RoboDK station: UR3_Pick_Place.rdk

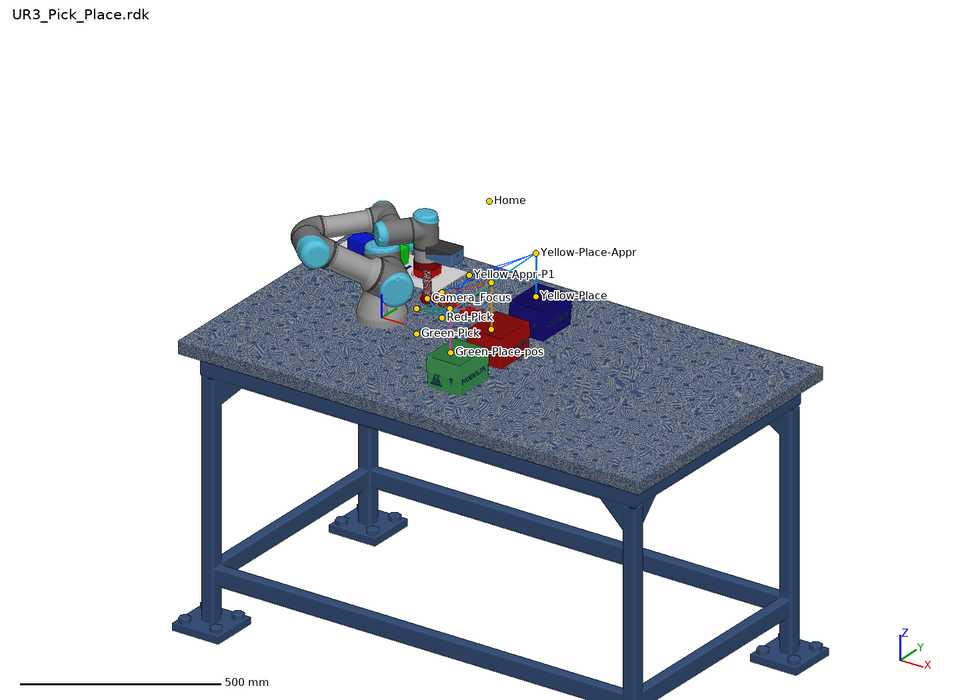
[picture v0: the station drawn from its stored meshes, robots at their saved joint values, targets as dots, program paths as lines]
Station UR3_Pick_Place (saved by RoboDK 5.4.1). Poses are relative to the parent item; angles as X-Y-Z fixed-axis rotations.
Station parameters (name, value as stored): IO_5, 1
  - frame UR3 Base at (0, 0, 0) mm
    - robot UR3: 6 axes, payload 3 kg, reach 500 mm, repeatability 0.1 mm, weight 11 kg
        modified DH rows (alpha deg, a mm, theta deg, d mm): 0, 0, 0, 151.9; 90, 0, 180, 0; 0, 243.65, 0, 0; 0, 213, 0, 110.4; -90, 0, 0, 83.4; 90, 0, 180, 82.4
        joint limits [-360, -360, -360, -360, -360, -360] to [360, 360, 360, 360, 360, 360]; home [0, -90, -90, 0, 90, 0]; saved at [48.153, -30.635, -146.156, -92.197, 88.87, 48.143]
      - tool Suction_Gripper, TCP at (0, 0, 110) mm, size 63.3 x 62.3 x 118 mm, geometry from Suction_Gripper.STEP
      - tool Camera, TCP at (0.03, -70.24, -12.53) mm, size 53 x 116 x 38 mm, geometry from Cam2D_SICK_VSPP_5F2113.sld
    - target Home (Cartesian target) at (403.4, -110.4, 478.95) mm, rotated rx -90 ry 0 rz -90 deg; joints [0, -90, -90, 0, 90, 0] of UR3
    - target Camera_Focus (Cartesian target) at (144.98, -9.29, 97.12) mm, rotated rx -178.48 ry 0 rz -90 deg; joints [48.127, -30.627, -146.695, -91.665, 88.87, 48.117] of UR3
    - target Yellow-Pick (Cartesian target) at (193.61, 104.25, 59.99) mm, rotated rx -179.29 ry 0 rz -90 deg; joints [59.044, -76.454, -144.258, -48.925, 89.395, 59.042] of UR3
    - target Yellow-Appr-P1 (Cartesian target) at (193.61, 104.25, 129.98) mm, rotated rx -179.29 ry 0 rz -90 deg; joints [59.044, -65.301, -129.223, -75.113, 89.395, 59.042] of UR3
    - target Yellow-Place (Cartesian target) at (346.96, 173.82, 85.56) mm, rotated rx -179.29 ry 0 rz -90 deg; joints [43.387, -113.771, -94.131, -61.585, 89.515, 43.384] of UR3
    - target Yellow-Place-Appr (Cartesian target) at (346.96, 173.82, 205.56) mm, rotated rx -179.29 ry 0 rz -90 deg; joints [43.389, -107.639, -68.833, -93.015, 89.515, 43.387] of UR3
    - target Red-Pick (Cartesian target) at (194.79, -15.82, 59.73) mm, rotated rx -179.29 ry 0 rz -90 deg; joints [30.172, -66.701, -149.718, -52.971, 89.645, 30.171] of UR3
    - target Red-Appr (Cartesian target) at (194.8, -15.82, 129.73) mm, rotated rx -179.29 ry 0 rz -90 deg; joints [30.173, -56.356, -133.241, -79.793, 89.645, 30.171] of UR3
    - target Red-Place-Appr (Cartesian target) at (344.8, -15.82, 199.73) mm, rotated rx -179.29 ry 0 rz -90 deg; joints [16.143, -96.634, -84.116, -88.571, 89.804, 16.142] of UR3
    - target Red-Place (Cartesian target) at (344.8, -15.82, 69.73) mm, rotated rx -179.29 ry 0 rz -90 deg; joints [16.142, -106.602, -109.753, -52.967, 89.804, 16.141] of UR3
    - target Green-Pick (Cartesian target) at (194.8, -125.82, 59.73) mm, rotated rx -179.29 ry 0 rz -90 deg; joints [-4.48, -80.711, -141.556, -47.028, 90.055, -4.48] of UR3
    - target Green-pick-aapr (Cartesian target) at (194.8, -125.82, 129.73) mm, rotated rx -179.29 ry 0 rz -90 deg; joints [-4.48, -69.374, -127.223, -72.7, 90.055, -4.48] of UR3
    - target Green-Place-pos (Cartesian target) at (348.16, -199.1, 80.31) mm, rotated rx -179.29 ry 0 rz -90 deg; joints [-13.869, -117.211, -90.452, -61.652, 90.169, -13.868] of UR3
    - target Green-place-appr (Cartesian target) at (344.79, -195.82, 199.73) mm, rotated rx -179.29 ry 0 rz -90 deg; joints [-13.51, -109.8, -67.516, -91.997, 90.165, -13.509] of UR3
    - object RoboDK Nametag Plate 500x200mm at (30, 330, 0) mm, rotated rx 0 ry 0 rz 90 deg, size 140 x 350 x 3.5 mm, geometry from RoboDK-Nametag-Plate-500x200mm.sld
  - object Table 1400x800x800 at (0, 0, 0) mm, size 1420 x 820 x 800 mm, geometry from Table-1400mmx800mmx800mm.sld
  - program Prog_Place_Blue (11 instructions, listed below)
  - program Prog_Place_Red (9 instructions, listed below)
  - program Prog_Place_Green (10 instructions, listed below)
  - camera Camera
  - program Prog_Return_Green (9 instructions, listed below)
  - program Prog_Return_Red (10 instructions, listed below)
  - program Prog_Return_Blue (8 instructions, listed below)
  - program Program_Animation (6 instructions, listed below)
  - object Blue-Box at (307.84, 115.7, 0) mm, size 109.7 x 131.2 x 86.2 mm, geometry from Box-12inx10in-Opened.sld
  - object Red-Box at (313.37, -73.28, 0) mm, size 109.7 x 131.2 x 86.2 mm, geometry from Box-12inx10in-Opened.sld
  - object Green-Box at (316.63, -256.72, 0) mm, size 109.7 x 131.2 x 86.2 mm, geometry from Box-12inx10in-Opened.sld
  - object Red-Cube at (-70, 237, 0) mm, size 50 x 50 x 50 mm, geometry from Cube-50mm.sld
  - object Blue-Cube at (-270, 237, 0) mm, size 50 x 50 x 50 mm, geometry from Cube-50mm.sld
  - object Green-Cube at (-170, 237, 0) mm, size 50 x 50 x 50 mm, geometry from Cube-50mm.sld
  - camera Camera 2
  - program Prog_Home_Pos (3 instructions, listed below)
  - program Prog_Cam_Pos (3 instructions, listed below)
  - object IDLEArea at (-40, 380, 0) mm, rotated rx 0 ry 0 rz 180 deg, size 181.5 x 27.8 x 8.8 mm, geometry from IDLEArea.STEP
  - object WorkArea at (280, 160, 0) mm, rotated rx 0 ry 0 rz 180 deg, size 271.5 x 30 x 9 mm, geometry from WorkArea.STEP
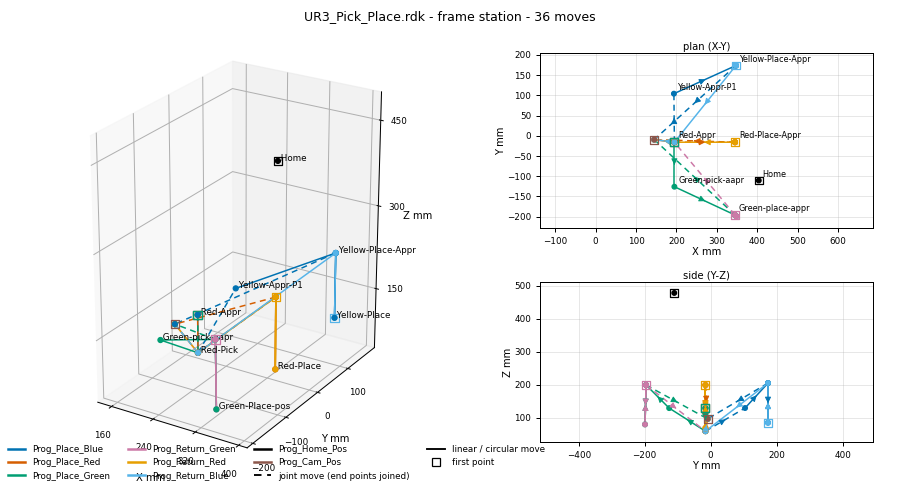
[picture p0: tool path of UR3_Pick_Place.rdk in frame station, 36 of 36 moves have a stored position in this frame; points joined in program order, loops and branches not executed]

--- program Prog_Place_Blue (robot UR3) ---
  Set Ref.: UR3 Base
  Set Tool: Gripper at (0, 0, 108) mm
  MoveJ (Red-Appr)
  MoveL (Red-Pick)
  Attach to Suction_Gripper
  MoveJ (Yellow-Appr-P1)
  MoveL (Yellow-Place-Appr)
  MoveL (Yellow-Place)
  Detach from Suction_Gripper
  MoveL (Yellow-Place-Appr)
  MoveJ (Camera_Focus)

--- program Prog_Place_Red (robot UR3) ---
  Set Ref.: UR3 Base
  MoveL (Red-Appr)
  MoveL (Red-Pick)
  Attach to Suction_Gripper
  MoveJ (Red-Place-Appr)
  MoveL (Red-Place)
  Detach from Suction_Gripper
  MoveL (Red-Place-Appr)
  MoveJ (Camera_Focus)

--- program Prog_Place_Green (robot UR3) ---
  Set Ref.: UR3 Base
  MoveL (Red-Appr)
  MoveJ (Red-Pick)
  Attach to Suction_Gripper
  MoveL (Green-pick-aapr)
  MoveL (Green-place-appr)
  MoveL (Green-Place-pos)
  Detach from Suction_Gripper
  MoveL (Green-place-appr)
  MoveJ (Camera_Focus)

--- program Prog_Return_Green (robot UR3) ---
  Set Ref.: UR3 Base
  Set Tool: Suction_Gripper
  MoveJ (Green-place-appr)
  MoveL (Green-Place-pos)
  Attach to Suction_Gripper
  MoveL (Green-place-appr)
  MoveJ (Red-Pick)
  Detach from Suction_Gripper
  MoveL (Camera_Focus)

--- program Prog_Return_Red (robot UR3) ---
  Set Ref.: UR3 Base
  Set Tool: Suction_Gripper
  MoveJ (Red-Place-Appr)
  MoveL (Red-Place)
  Attach to Suction_Gripper
  MoveL (Red-Place-Appr)
  MoveL (Red-Pick)
  Detach from Suction_Gripper
  MoveL (Camera_Focus)
  Set IO_5=1

--- program Prog_Return_Blue (robot UR3) ---
  Set Ref.: UR3 Base
  Set Tool: Suction_Gripper
  MoveJ (Yellow-Place)
  Attach to Suction_Gripper
  MoveL (Yellow-Place-Appr)
  MoveL (Red-Pick)
  Detach from Suction_Gripper
  MoveJ (Camera_Focus)

--- program Program_Animation (robot UR3) ---
  Call Prog1
  Call Prog2
  Call Prog3
  Call Prog4
  Call Prog5
  Call Prog6

--- program Prog_Home_Pos (robot UR3) ---
  Set Ref.: UR3 Base
  Set Tool: Suction_Gripper
  MoveL (Home)

--- program Prog_Cam_Pos (robot UR3) ---
  Set Ref.: UR3 Base
  Set Tool: Suction_Gripper
  MoveL (Camera_Focus)
